Yaskawa INFORM job: DEMO_NAIHAN_0625_2_TOOL0.JBI

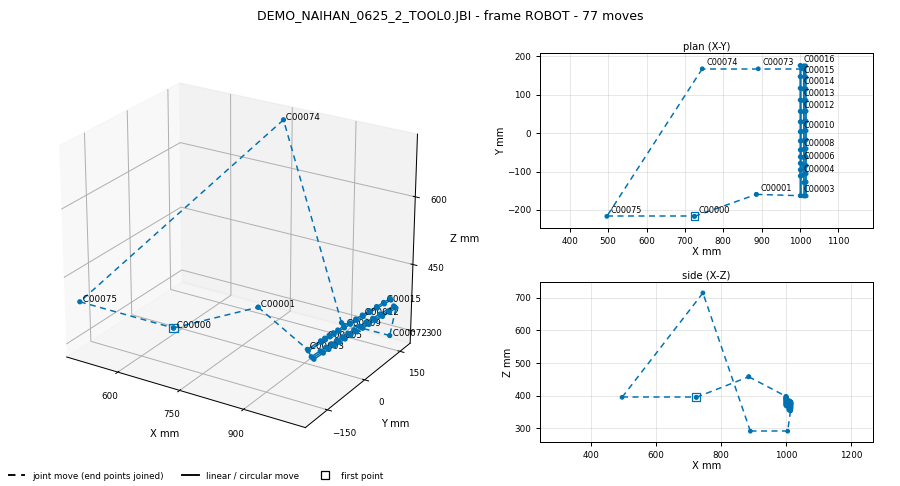
[picture p0: tool path of DEMO_NAIHAN_0625_2_TOOL0.JBI in frame ROBOT, 77 of 77 moves have a stored position in this frame; points joined in program order, loops and branches not executed]
/JOB
//NAME DEMO_NAIHAN_SIDE_0625_2_TOOL0
//POS
///NPOS 77,0,0,0,0,0
///TOOL 0
///USER 0
///POSTYPE ROBOT
///RECTAN
///RCONF 1,0,0,0,0,0,0,0,0,0,0,0,0,0,0,0,0,0,0,0,0,0,0,0
C00000=724.889,-216.680,394.500,-180.000,-0.000,-0.000
///USER 0
///POSTYPE ROBOT
///RECTAN
///RCONF 0,0,0,0,0,0,0,0,0,0,0,0,0,0,0,0,0,0,0,0,0,0,0,0
C00001=886.160,-159.406,457.717,-85.028,-4.406,-90.070
C00002=886.160,-159.406,457.717,-85.028,-4.406,-90.070
C00003=1000.375,-162.892,397.610,-85.032,-3.708,-90.010
C00004=1000.373,-111.597,394.487,-85.032,-3.708,-90.010
C00005=1000.373,-95.500,393.443,-85.016,-3.886,-90.010
C00006=1000.374,-78.358,392.278,-85.028,-4.069,-90.009
C00007=1000.371,-61.619,391.087,-85.066,-4.228,-90.001
C00008=1000.370,-43.509,389.748,-85.148,-4.435,-89.992
C00009=1000.363,-20.297,387.948,-85.293,-4.638,-89.969
C00010=1000.347,3.823,385.991,-85.516,-4.820,-89.938
C00011=1000.316,29.650,383.813,-85.849,-4.991,-89.899
C00012=1000.267,56.924,381.431,-86.305,-5.133,-89.856
C00013=1000.200,86.172,378.804,-86.928,-5.261,-89.817
C00014=1000.119,117.153,375.952,-87.747,-5.370,-89.794
C00015=1000.040,147.317,373.118,-88.707,-5.685,-89.811
C00016=999.971,176.185,370.245,-88.707,-5.685,-89.811
C00017=1002.013,175.921,367.556,-88.707,-5.685,-89.811
C00018=1002.111,147.056,370.452,-88.708,-5.272,-89.801
C00019=1002.219,116.895,373.308,-87.747,-5.222,-89.788
C00020=1002.325,85.923,376.178,-86.928,-5.164,-89.811
C00021=1002.410,56.691,378.819,-86.305,-5.056,-89.851
C00022=1002.471,29.425,381.209,-85.849,-4.928,-89.895
C00023=1002.509,3.609,383.394,-85.516,-4.781,-89.935
C00024=1002.531,-20.500,385.354,-85.293,-4.628,-89.968
C00025=1002.542,-43.703,387.158,-85.148,-4.463,-89.995
C00026=1002.545,-61.813,388.499,-85.066,-4.321,-90.009
C00027=1002.546,-78.542,389.688,-85.027,-4.201,-90.020
C00028=1002.546,-95.671,390.851,-85.015,-4.078,-90.027
C00029=1002.545,-111.757,391.894,-85.031,-3.977,-90.033
C00030=1002.548,-163.054,395.017,-85.082,-3.945,-90.044
C00031=1009.722,-163.599,384.381,-85.080,-4.129,-90.060
C00032=1009.722,-128.751,382.326,-31.715,-3.450,-90.069
C00033=1009.727,-107.125,380.988,-31.695,-3.705,-90.070
C00034=1009.732,-85.811,379.574,-31.674,-3.955,-90.065
C00035=1009.734,-63.934,378.025,-31.653,-4.207,-90.052
C00036=1009.732,-41.954,376.371,-31.632,-4.452,-90.033
C00037=1009.722,-18.867,374.536,-31.612,-4.691,-90.005
C00038=1009.700,5.110,372.529,-31.592,-4.920,-89.964
C00039=1009.661,29.831,370.362,-31.574,-5.130,-89.915
C00040=1009.598,55.930,367.980,-31.558,-5.331,-89.868
C00041=1009.508,84.324,365.290,-31.541,-5.526,-89.824
C00042=1009.390,114.344,362.345,-31.525,-5.710,-89.789
C00043=1009.121,174.973,356.208,-31.516,-5.848,-89.704
C00044=1011.487,175.236,354.677,-31.516,-5.848,-89.704
C00045=1012.511,145.654,357.169,-31.604,-5.293,-88.804
C00046=1012.625,115.245,360.260,-31.547,-5.580,-89.569
C00047=1012.730,85.244,363.213,-31.556,-5.433,-89.663
C00048=1012.810,57.503,365.850,-31.569,-5.263,-89.740
C00049=1012.866,31.400,368.242,-31.581,-5.083,-89.817
C00050=1012.901,6.655,370.420,-31.597,-4.890,-89.894
C00051=1012.921,-17.272,372.430,-31.613,-4.684,-89.967
C00052=1012.928,-40.395,374.276,-31.631,-4.469,-90.035
C00053=1012.928,-62.349,375.935,-31.648,-4.252,-90.099
C00054=1012.924,-84.167,377.487,-31.666,-4.032,-90.162
C00055=1012.918,-105.581,378.914,-31.683,-3.814,-90.222
C00056=1012.913,-127.211,380.259,-31.701,-3.601,-90.289
C00057=1012.912,-163.368,382.396,-31.687,-3.723,-90.622
C00058=1015.786,-163.473,380.609,-31.687,-3.724,-90.623
C00059=1015.795,-127.321,378.484,-31.714,-3.465,-90.069
C00060=1015.800,-105.699,377.141,-31.693,-3.722,-90.073
C00061=1015.807,-84.292,375.716,-31.672,-3.975,-90.070
C00062=1015.812,-62.481,374.164,-31.651,-4.227,-90.058
C00063=1015.813,-40.534,372.508,-31.631,-4.471,-90.038
C00064=1015.806,-17.418,370.664,-31.610,-4.711,-90.012
C00065=1015.787,6.505,368.654,-31.590,-4.939,-89.974
C00066=1015.753,31.247,366.478,-31.571,-5.151,-89.930
C00067=1015.698,57.345,364.088,-31.555,-5.352,-89.884
C00068=1015.618,85.083,361.450,-31.539,-5.545,-89.845
C00069=1015.513,115.079,358.499,-31.522,-5.736,-89.825
C00070=1015.399,145.489,355.409,-31.663,-4.886,-88.140
C00071=1014.427,175.184,352.858,-31.662,-4.889,-88.138
C00072=1005.856,167.678,290.346,-31.576,-5.475,-89.093
C00073=891.077,167.678,290.346,-31.576,-5.475,-89.093
C00074=745.180,167.678,715.406,-31.576,-5.475,-89.093
///USER 0
///POSTYPE ROBOT
///RECTAN
///RCONF 1,0,0,0,0,0,0,0,0,0,0,0,0,0,0,0,0,0,0,0,0,0,0,0
C00075=496.664,-216.680,394.500,-180.000,-0.000,-0.000
C00076=724.889,-216.680,394.500,-180.000,-0.000,-0.000
//INST
///DATE 2021/06/25 12:19
///ATTR SC,RW,RJ
////FRAME ROBOT
///GROUP1 RB1
NOP
MOVJ C00000 VJ=25.00 PL=0
MOVJ C00001 VJ=25.00 PL=0
'Path Start: naihan
MOVJ C00002 VJ=25.00 PL=0
MOVJ C00003 VJ=25.00 PL=0
SPYON
MOVL C00004 V=800.0 PL=8
MOVL C00005 V=800.0 PL=8
MOVL C00006 V=800.0 PL=8
MOVL C00007 V=800.0 PL=8
MOVL C00008 V=800.0 PL=8
MOVL C00009 V=800.0 PL=8
MOVL C00010 V=800.0 PL=8
MOVL C00011 V=800.0 PL=8
MOVL C00012 V=800.0 PL=8
MOVL C00013 V=800.0 PL=8
MOVL C00014 V=800.0 PL=8
MOVL C00015 V=800.0 PL=8
MOVL C00016 V=800.0 PL=0
SPYOF
MOVJ C00017 VJ=25.00 PL=0
SPYON
MOVL C00018 V=800.0 PL=8
MOVL C00019 V=800.0 PL=8
MOVL C00020 V=800.0 PL=8
MOVL C00021 V=800.0 PL=8
MOVL C00022 V=800.0 PL=8
MOVL C00023 V=800.0 PL=8
MOVL C00024 V=800.0 PL=8
MOVL C00025 V=800.0 PL=8
MOVL C00026 V=800.0 PL=8
MOVL C00027 V=800.0 PL=8
MOVL C00028 V=800.0 PL=8
MOVL C00029 V=800.0 PL=8
MOVL C00030 V=800.0 PL=0
SPYOF
MOVJ C00031 VJ=25.00 PL=0
SPYON
MOVL C00032 V=800.0 PL=8
MOVL C00033 V=800.0 PL=8
MOVL C00034 V=800.0 PL=8
MOVL C00035 V=800.0 PL=8
MOVL C00036 V=800.0 PL=8
MOVL C00037 V=800.0 PL=8
MOVL C00038 V=800.0 PL=8
MOVL C00039 V=800.0 PL=8
MOVL C00040 V=800.0 PL=8
MOVL C00041 V=800.0 PL=8
MOVL C00042 V=800.0 PL=8
MOVL C00043 V=800.0 PL=0
SPYOF
MOVJ C00044 VJ=25.00 PL=0
SPYON
MOVL C00045 V=800.0 PL=8
MOVL C00046 V=800.0 PL=8
MOVL C00047 V=800.0 PL=8
MOVL C00048 V=800.0 PL=8
MOVL C00049 V=800.0 PL=8
MOVL C00050 V=800.0 PL=8
MOVL C00051 V=800.0 PL=8
MOVL C00052 V=800.0 PL=8
MOVL C00053 V=800.0 PL=8
MOVL C00054 V=800.0 PL=8
MOVL C00055 V=800.0 PL=8
MOVL C00056 V=800.0 PL=8
MOVL C00057 V=800.0 PL=0
SPYOF
MOVJ C00058 VJ=25.00 PL=0
SPYON
MOVL C00059 V=800.0 PL=8
MOVL C00060 V=800.0 PL=8
MOVL C00061 V=800.0 PL=8
MOVL C00062 V=800.0 PL=8
MOVL C00063 V=800.0 PL=8
MOVL C00064 V=800.0 PL=8
MOVL C00065 V=800.0 PL=8
MOVL C00066 V=800.0 PL=8
MOVL C00067 V=800.0 PL=8
MOVL C00068 V=800.0 PL=8
MOVL C00069 V=800.0 PL=8
MOVL C00070 V=800.0 PL=8
MOVL C00071 V=800.0 PL=0
SPYOF
MOVJ C00072 VJ=25.00 PL=0
MOVJ C00073 VJ=25.00 PL=0
MOVJ C00074 VJ=25.00 PL=0
'Path End
MOVJ C00075 VJ=25.00 PL=0
MOVJ C00076 VJ=25.00 PL=0
END
